// TIA Portal V17 export
// export: Created 2025-03-07T09:18:45.8638249Z, ExportSetting WithDefaults, DisplayName Totally Integrated Automation Portal, DisplayVersion V17 Update 8, DisplayName TIA Portal Openness, DisplayVersion V17 Update 8, DisplayName TIA Portal Version Control Interface, DisplayVersion V17, DisplayName SINAMICS Startdrive Advanced, DisplayVersion V17 SP2, DisplayName SINAMICS Startdrive G110M, G120, G120C, G120D, G120P, G115D, DisplayVersion V17 SP2, DisplayName SINAMICS Startdrive G130, G150, S120, S150, SINAMICS MV, S210, DisplayVersion V17 SP2, DisplayName STEP 7 Professional, DisplayVersion V17 Update 8, DisplayName SINUMERIK ONE STEP 7 Toolbox, DisplayVersion V17 Update 12, DisplayName SINUMERIK 840D sl STEP 7 Toolbox, DisplayVersion V17 Update 12, DisplayName STEP 7 Safety, DisplayVersion V17 Update 6, DisplayName WinCC Advanced, DisplayVersion V17 Update 8
FUNCTION "FC2391_SAVE_ENERGY" : Void   // FC2391, LAD
{ S7_Optimized_Access := 'FALSE' }
AUTHOR : ETXETAR
VERSION : 1.0
// stored: AutoNumber false, IsIECCheckEnabled false, SetENOAutomatically false, UDAEnableTagReadback false
   VAR_TEMP
      O_BYTE_0 : Struct   // OPTIONS BYTE 0
         AUTO_RECOVERY : Bool;   // AUTO RECOVERY OPTION
         RUNOUT : Bool;   // RUNOUT OPTION
      END_STRUCT;
   END_VAR
   VAR CONSTANT
      FC_NUMBER : DInt := 2391;
   END_VAR
   VAR_TEMP   // added for the SCL form of the ladder/FBD networks
      _w1 : Bool;
   END_VAR
BEGIN

REGION Network 1: OPTIONS OFF
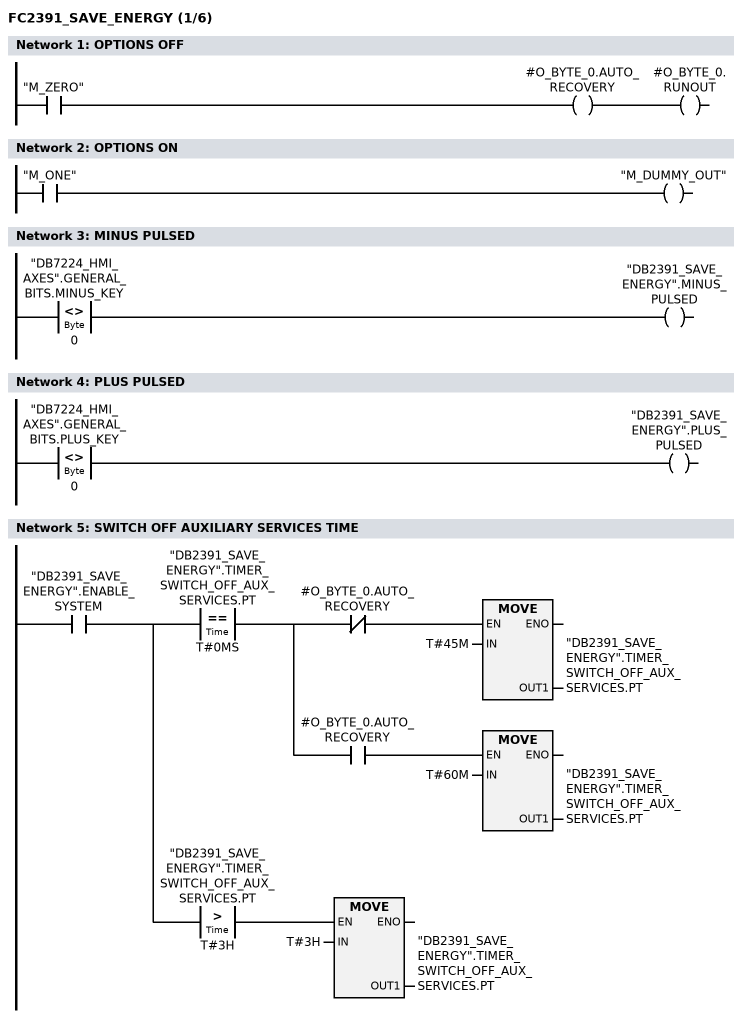
   RUNG wire#powerrail
      Contact( "M_ZERO" )
      Coil( #O_BYTE_0.AUTO_RECOVERY )
      Coil( #O_BYTE_0.RUNOUT )
   END_RUNG
   // the same network as SCL:
   #O_BYTE_0.AUTO_RECOVERY := "M_ZERO";
   #O_BYTE_0.RUNOUT := "M_ZERO";
END_REGION

REGION Network 2: OPTIONS ON
   RUNG wire#powerrail
      Contact( "M_ONE" )
      Coil( "M_DUMMY_OUT" )
   END_RUNG
   // the same network as SCL:
   "M_DUMMY_OUT" := "M_ONE";
END_REGION

REGION Network 3: MINUS PULSED
   RUNG wire#powerrail
      { S7_Templates := "SrcType := Byte" } NE_Contact(in1 := "DB7224_HMI_AXES".GENERAL_BITS.MINUS_KEY, in2 := 0)
      Coil( "DB2391_SAVE_ENERGY".MINUS_PULSED )
   END_RUNG
   // the same network as SCL:
   "DB2391_SAVE_ENERGY".MINUS_PULSED := "DB7224_HMI_AXES".GENERAL_BITS.MINUS_KEY <> 0;
END_REGION

REGION Network 4: PLUS PULSED
   RUNG wire#powerrail
      { S7_Templates := "SrcType := Byte" } NE_Contact(in1 := "DB7224_HMI_AXES".GENERAL_BITS.PLUS_KEY, in2 := 0)
      Coil( "DB2391_SAVE_ENERGY".PLUS_PULSED )
   END_RUNG
   // the same network as SCL:
   "DB2391_SAVE_ENERGY".PLUS_PULSED := "DB7224_HMI_AXES".GENERAL_BITS.PLUS_KEY <> 0;
END_REGION

REGION Network 5: SWITCH OFF AUXILIARY SERVICES TIME
   RUNG wire#powerrail
      Contact( "DB2391_SAVE_ENERGY".ENABLE_SYSTEM )
      wire#w1
      { S7_Templates := "SrcType := Time" } EQ_Contact(in1 := "DB2391_SAVE_ENERGY".TIMER_SWITCH_OFF_AUX_SERVICES.PT, in2 := T#0MS)
      wire#w2
      I_Contact( #O_BYTE_0.AUTO_RECOVERY )
      { S7_GenerateENO := "TRUE" } Move(in := T#45M, out1 => "DB2391_SAVE_ENERGY".TIMER_SWITCH_OFF_AUX_SERVICES.PT)
   END_RUNG
   RUNG wire#w2
      Contact( #O_BYTE_0.AUTO_RECOVERY )
      { S7_GenerateENO := "TRUE" } Move(in := T#60M, out1 => "DB2391_SAVE_ENERGY".TIMER_SWITCH_OFF_AUX_SERVICES.PT)
   END_RUNG
   RUNG wire#w1
      { S7_Templates := "SrcType := Time" } GT_Contact(in1 := "DB2391_SAVE_ENERGY".TIMER_SWITCH_OFF_AUX_SERVICES.PT, in2 := T#3H)
      { S7_GenerateENO := "TRUE" } Move(in := T#3H, out1 => "DB2391_SAVE_ENERGY".TIMER_SWITCH_OFF_AUX_SERVICES.PT)
   END_RUNG
   // the same network as SCL:
   #_w1 := "DB2391_SAVE_ENERGY".ENABLE_SYSTEM AND ("DB2391_SAVE_ENERGY".TIMER_SWITCH_OFF_AUX_SERVICES.PT = T#0MS);
   IF #_w1 AND NOT #O_BYTE_0.AUTO_RECOVERY THEN
       "DB2391_SAVE_ENERGY".TIMER_SWITCH_OFF_AUX_SERVICES.PT := T#45M;
   END_IF;
   IF #_w1 AND #O_BYTE_0.AUTO_RECOVERY THEN
       "DB2391_SAVE_ENERGY".TIMER_SWITCH_OFF_AUX_SERVICES.PT := T#60M;
   END_IF;
   IF "DB2391_SAVE_ENERGY".ENABLE_SYSTEM AND ("DB2391_SAVE_ENERGY".TIMER_SWITCH_OFF_AUX_SERVICES.PT > T#3H) THEN
       "DB2391_SAVE_ENERGY".TIMER_SWITCH_OFF_AUX_SERVICES.PT := T#3H;
   END_IF;
END_REGION

REGION Network 6: SWITCH OFF MAIN SERVICES TIME
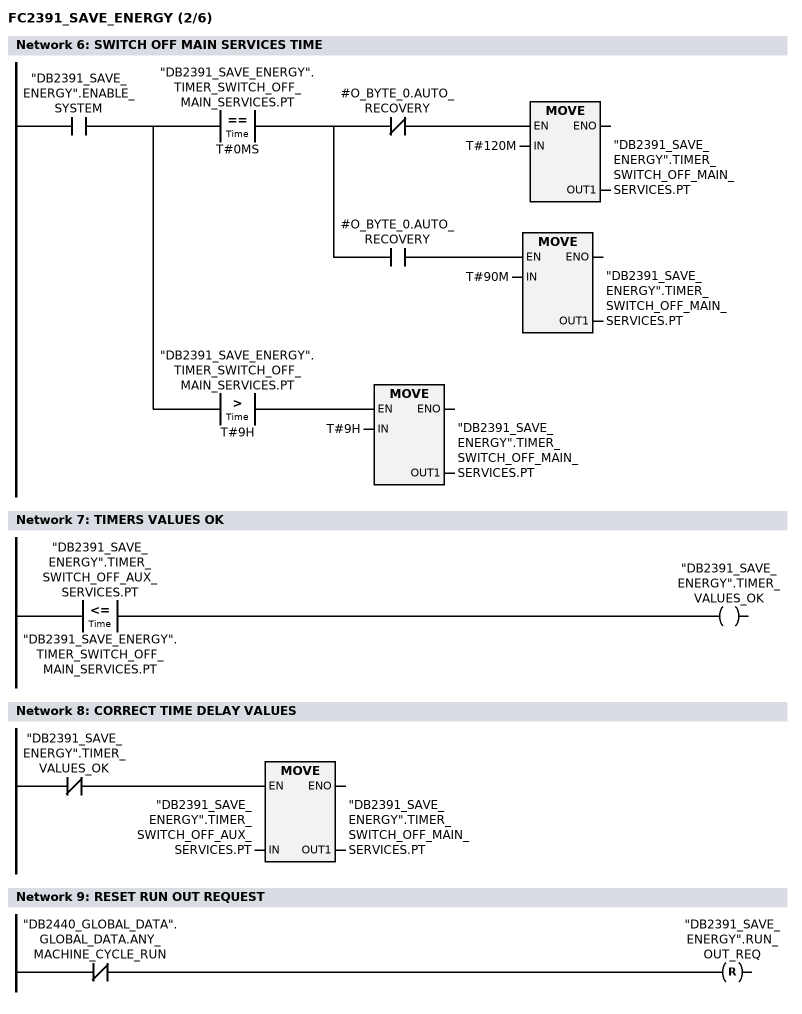
   RUNG wire#powerrail
      Contact( "DB2391_SAVE_ENERGY".ENABLE_SYSTEM )
      wire#w1
      { S7_Templates := "SrcType := Time" } EQ_Contact(in1 := "DB2391_SAVE_ENERGY".TIMER_SWITCH_OFF_MAIN_SERVICES.PT, in2 := T#0MS)
      wire#w2
      I_Contact( #O_BYTE_0.AUTO_RECOVERY )
      { S7_GenerateENO := "TRUE" } Move(in := T#120M, out1 => "DB2391_SAVE_ENERGY".TIMER_SWITCH_OFF_MAIN_SERVICES.PT)
   END_RUNG
   RUNG wire#w2
      Contact( #O_BYTE_0.AUTO_RECOVERY )
      { S7_GenerateENO := "TRUE" } Move(in := T#90M, out1 => "DB2391_SAVE_ENERGY".TIMER_SWITCH_OFF_MAIN_SERVICES.PT)
   END_RUNG
   RUNG wire#w1
      { S7_Templates := "SrcType := Time" } GT_Contact(in1 := "DB2391_SAVE_ENERGY".TIMER_SWITCH_OFF_MAIN_SERVICES.PT, in2 := T#9H)
      { S7_GenerateENO := "TRUE" } Move(in := T#9H, out1 => "DB2391_SAVE_ENERGY".TIMER_SWITCH_OFF_MAIN_SERVICES.PT)
   END_RUNG
   // the same network as SCL:
   #_w1 := "DB2391_SAVE_ENERGY".ENABLE_SYSTEM AND ("DB2391_SAVE_ENERGY".TIMER_SWITCH_OFF_MAIN_SERVICES.PT = T#0MS);
   IF #_w1 AND NOT #O_BYTE_0.AUTO_RECOVERY THEN
       "DB2391_SAVE_ENERGY".TIMER_SWITCH_OFF_MAIN_SERVICES.PT := T#120M;
   END_IF;
   IF #_w1 AND #O_BYTE_0.AUTO_RECOVERY THEN
       "DB2391_SAVE_ENERGY".TIMER_SWITCH_OFF_MAIN_SERVICES.PT := T#90M;
   END_IF;
   IF "DB2391_SAVE_ENERGY".ENABLE_SYSTEM AND ("DB2391_SAVE_ENERGY".TIMER_SWITCH_OFF_MAIN_SERVICES.PT > T#9H) THEN
       "DB2391_SAVE_ENERGY".TIMER_SWITCH_OFF_MAIN_SERVICES.PT := T#9H;
   END_IF;
END_REGION

REGION Network 7: TIMERS VALUES OK
   RUNG wire#powerrail
      { S7_Templates := "SrcType := Time" } LE_Contact(in1 := "DB2391_SAVE_ENERGY".TIMER_SWITCH_OFF_AUX_SERVICES.PT, in2 := "DB2391_SAVE_ENERGY".TIMER_SWITCH_OFF_MAIN_SERVICES.PT)
      Coil( "DB2391_SAVE_ENERGY".TIMER_VALUES_OK )
   END_RUNG
   // the same network as SCL:
   "DB2391_SAVE_ENERGY".TIMER_VALUES_OK := "DB2391_SAVE_ENERGY".TIMER_SWITCH_OFF_AUX_SERVICES.PT <= "DB2391_SAVE_ENERGY".TIMER_SWITCH_OFF_MAIN_SERVICES.PT;
END_REGION

REGION Network 8: CORRECT TIME DELAY VALUES
   RUNG wire#powerrail
      I_Contact( "DB2391_SAVE_ENERGY".TIMER_VALUES_OK )
      Move(in := "DB2391_SAVE_ENERGY".TIMER_SWITCH_OFF_AUX_SERVICES.PT, out1 => "DB2391_SAVE_ENERGY".TIMER_SWITCH_OFF_MAIN_SERVICES.PT)
   END_RUNG
   // the same network as SCL:
   IF NOT "DB2391_SAVE_ENERGY".TIMER_VALUES_OK THEN
       "DB2391_SAVE_ENERGY".TIMER_SWITCH_OFF_MAIN_SERVICES.PT := "DB2391_SAVE_ENERGY".TIMER_SWITCH_OFF_AUX_SERVICES.PT;
   END_IF;
END_REGION

REGION Network 9: RESET RUN OUT REQUEST
   RUNG wire#powerrail
      I_Contact( "DB2440_GLOBAL_DATA".GLOBAL_DATA.ANY_MACHINE_CYCLE_RUN )
      R_Coil( "DB2391_SAVE_ENERGY".RUN_OUT_REQ )
   END_RUNG
   // the same network as SCL:
   IF NOT "DB2440_GLOBAL_DATA".GLOBAL_DATA.ANY_MACHINE_CYCLE_RUN THEN
       "DB2391_SAVE_ENERGY".RUN_OUT_REQ := FALSE;
   END_IF;
END_REGION

REGION Network 10: RUN OUT REQUEST
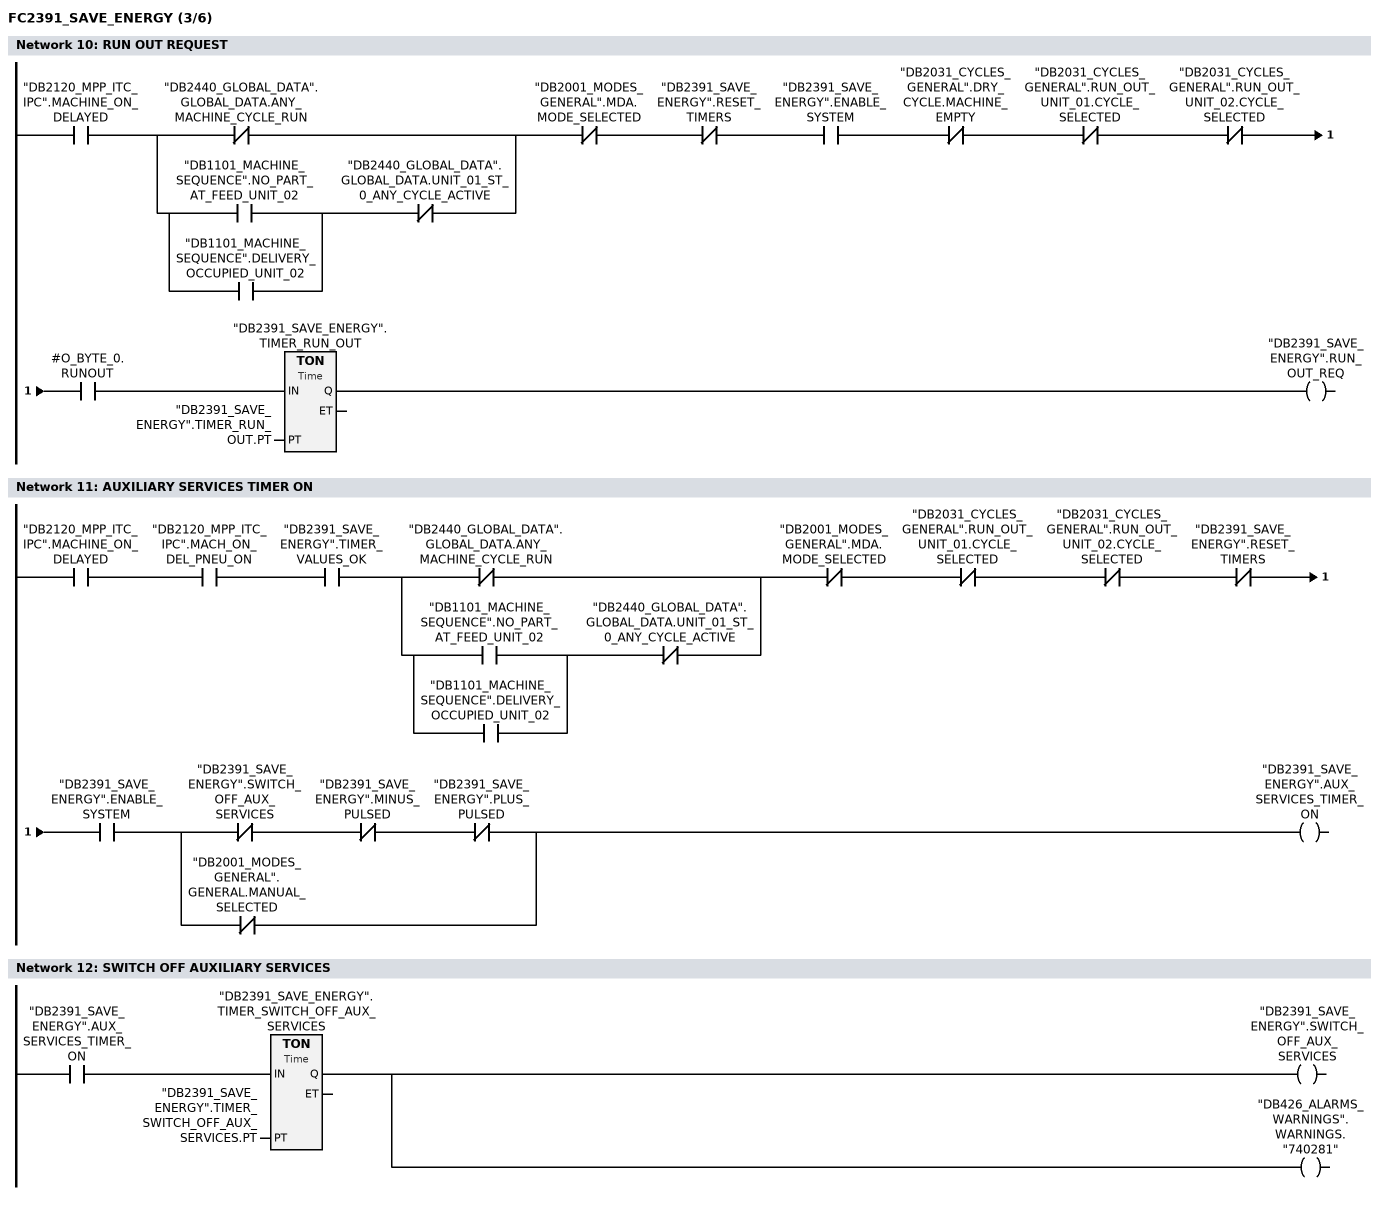
   RUNG wire#powerrail
      Contact( "DB2120_MPP_ITC_IPC".MACHINE_ON_DELAYED )
      wire#w1
      I_Contact( "DB2440_GLOBAL_DATA".GLOBAL_DATA.ANY_MACHINE_CYCLE_RUN )
      wire#w2
      I_Contact( "DB2001_MODES_GENERAL".MDA.MODE_SELECTED )
      I_Contact( "DB2391_SAVE_ENERGY".RESET_TIMERS )
      Contact( "DB2391_SAVE_ENERGY".ENABLE_SYSTEM )
      I_Contact( "DB2031_CYCLES_GENERAL".DRY_CYCLE.MACHINE_EMPTY )
      I_Contact( "DB2031_CYCLES_GENERAL".RUN_OUT_UNIT_01.CYCLE_SELECTED )
      I_Contact( "DB2031_CYCLES_GENERAL".RUN_OUT_UNIT_02.CYCLE_SELECTED )
      Contact( #O_BYTE_0.RUNOUT )
      { S7_Templates := "time_type := Time" } "DB2391_SAVE_ENERGY".TIMER_RUN_OUT.TON(pt := "DB2391_SAVE_ENERGY".TIMER_RUN_OUT.PT, et =>)
      Coil( "DB2391_SAVE_ENERGY".RUN_OUT_REQ )
   END_RUNG
   RUNG wire#w1
      Contact( "DB1101_MACHINE_SEQUENCE".NO_PART_AT_FEED_UNIT_02 )
      wire#w3
      I_Contact( "DB2440_GLOBAL_DATA".GLOBAL_DATA.UNIT_01_ST_0_ANY_CYCLE_ACTIVE )
   END_RUNG wire#w2
   RUNG wire#w1
      Contact( "DB1101_MACHINE_SEQUENCE".DELIVERY_OCCUPIED_UNIT_02 )
   END_RUNG wire#w3
   // the same network as SCL:
   "DB2391_SAVE_ENERGY".TIMER_RUN_OUT.TON(IN := "DB2120_MPP_ITC_IPC".MACHINE_ON_DELAYED AND (NOT "DB2440_GLOBAL_DATA".GLOBAL_DATA.ANY_MACHINE_CYCLE_RUN OR (("DB1101_MACHINE_SEQUENCE".NO_PART_AT_FEED_UNIT_02 OR "DB1101_MACHINE_SEQUENCE".DELIVERY_OCCUPIED_UNIT_02) AND NOT "DB2440_GLOBAL_DATA".GLOBAL_DATA.UNIT_01_ST_0_ANY_CYCLE_ACTIVE)) AND NOT "DB2001_MODES_GENERAL".MDA.MODE_SELECTED AND NOT "DB2391_SAVE_ENERGY".RESET_TIMERS AND "DB2391_SAVE_ENERGY".ENABLE_SYSTEM AND NOT "DB2031_CYCLES_GENERAL".DRY_CYCLE.MACHINE_EMPTY AND NOT "DB2031_CYCLES_GENERAL".RUN_OUT_UNIT_01.CYCLE_SELECTED AND NOT "DB2031_CYCLES_GENERAL".RUN_OUT_UNIT_02.CYCLE_SELECTED AND #O_BYTE_0.RUNOUT,
                           PT := "DB2391_SAVE_ENERGY".TIMER_RUN_OUT.PT);
   "DB2391_SAVE_ENERGY".RUN_OUT_REQ := "DB2391_SAVE_ENERGY".TIMER_RUN_OUT.Q;
END_REGION

REGION Network 11: AUXILIARY SERVICES TIMER ON
   RUNG wire#powerrail
      Contact( "DB2120_MPP_ITC_IPC".MACHINE_ON_DELAYED )
      Contact( "DB2120_MPP_ITC_IPC".MACH_ON_DEL_PNEU_ON )
      Contact( "DB2391_SAVE_ENERGY".TIMER_VALUES_OK )
      wire#w1
      I_Contact( "DB2440_GLOBAL_DATA".GLOBAL_DATA.ANY_MACHINE_CYCLE_RUN )
      wire#w2
      I_Contact( "DB2001_MODES_GENERAL".MDA.MODE_SELECTED )
      I_Contact( "DB2031_CYCLES_GENERAL".RUN_OUT_UNIT_01.CYCLE_SELECTED )
      I_Contact( "DB2031_CYCLES_GENERAL".RUN_OUT_UNIT_02.CYCLE_SELECTED )
      I_Contact( "DB2391_SAVE_ENERGY".RESET_TIMERS )
      Contact( "DB2391_SAVE_ENERGY".ENABLE_SYSTEM )
      wire#w4
      I_Contact( "DB2391_SAVE_ENERGY".SWITCH_OFF_AUX_SERVICES )
      I_Contact( "DB2391_SAVE_ENERGY".MINUS_PULSED )
      I_Contact( "DB2391_SAVE_ENERGY".PLUS_PULSED )
      wire#w5
      Coil( "DB2391_SAVE_ENERGY".AUX_SERVICES_TIMER_ON )
   END_RUNG
   RUNG wire#w1
      Contact( "DB1101_MACHINE_SEQUENCE".NO_PART_AT_FEED_UNIT_02 )
      wire#w3
      I_Contact( "DB2440_GLOBAL_DATA".GLOBAL_DATA.UNIT_01_ST_0_ANY_CYCLE_ACTIVE )
   END_RUNG wire#w2
   RUNG wire#w1
      Contact( "DB1101_MACHINE_SEQUENCE".DELIVERY_OCCUPIED_UNIT_02 )
   END_RUNG wire#w3
   RUNG wire#w4
      I_Contact( "DB2001_MODES_GENERAL".GENERAL.MANUAL_SELECTED )
   END_RUNG wire#w5
   // the same network as SCL:
   "DB2391_SAVE_ENERGY".AUX_SERVICES_TIMER_ON := "DB2120_MPP_ITC_IPC".MACHINE_ON_DELAYED AND "DB2120_MPP_ITC_IPC".MACH_ON_DEL_PNEU_ON AND "DB2391_SAVE_ENERGY".TIMER_VALUES_OK AND (NOT "DB2440_GLOBAL_DATA".GLOBAL_DATA.ANY_MACHINE_CYCLE_RUN OR (("DB1101_MACHINE_SEQUENCE".NO_PART_AT_FEED_UNIT_02 OR "DB1101_MACHINE_SEQUENCE".DELIVERY_OCCUPIED_UNIT_02) AND NOT "DB2440_GLOBAL_DATA".GLOBAL_DATA.UNIT_01_ST_0_ANY_CYCLE_ACTIVE)) AND NOT "DB2001_MODES_GENERAL".MDA.MODE_SELECTED AND NOT "DB2031_CYCLES_GENERAL".RUN_OUT_UNIT_01.CYCLE_SELECTED AND NOT "DB2031_CYCLES_GENERAL".RUN_OUT_UNIT_02.CYCLE_SELECTED AND NOT "DB2391_SAVE_ENERGY".RESET_TIMERS AND "DB2391_SAVE_ENERGY".ENABLE_SYSTEM AND ((NOT "DB2391_SAVE_ENERGY".SWITCH_OFF_AUX_SERVICES AND NOT "DB2391_SAVE_ENERGY".MINUS_PULSED AND NOT "DB2391_SAVE_ENERGY".PLUS_PULSED) OR NOT "DB2001_MODES_GENERAL".GENERAL.MANUAL_SELECTED);
END_REGION

REGION Network 12: SWITCH OFF AUXILIARY SERVICES
   RUNG wire#powerrail
      Contact( "DB2391_SAVE_ENERGY".AUX_SERVICES_TIMER_ON )
      { S7_Templates := "time_type := Time" } "DB2391_SAVE_ENERGY".TIMER_SWITCH_OFF_AUX_SERVICES.TON(pt := "DB2391_SAVE_ENERGY".TIMER_SWITCH_OFF_AUX_SERVICES.PT, et =>)
      wire#w1
      Coil( "DB2391_SAVE_ENERGY".SWITCH_OFF_AUX_SERVICES )
   END_RUNG
   RUNG wire#w1
      Coil( "DB426_ALARMS_WARNINGS".WARNINGS."740281" )
   END_RUNG
   // the same network as SCL:
   "DB2391_SAVE_ENERGY".TIMER_SWITCH_OFF_AUX_SERVICES.TON(IN := "DB2391_SAVE_ENERGY".AUX_SERVICES_TIMER_ON,
                           PT := "DB2391_SAVE_ENERGY".TIMER_SWITCH_OFF_AUX_SERVICES.PT);
   "DB2391_SAVE_ENERGY".SWITCH_OFF_AUX_SERVICES := "DB2391_SAVE_ENERGY".TIMER_SWITCH_OFF_AUX_SERVICES.Q;
   "DB426_ALARMS_WARNINGS".WARNINGS."740281" := "DB2391_SAVE_ENERGY".TIMER_SWITCH_OFF_AUX_SERVICES.Q;
END_REGION

REGION Network 13: SWTICH OFF AUXILIARY SERVICES TIME LEFT
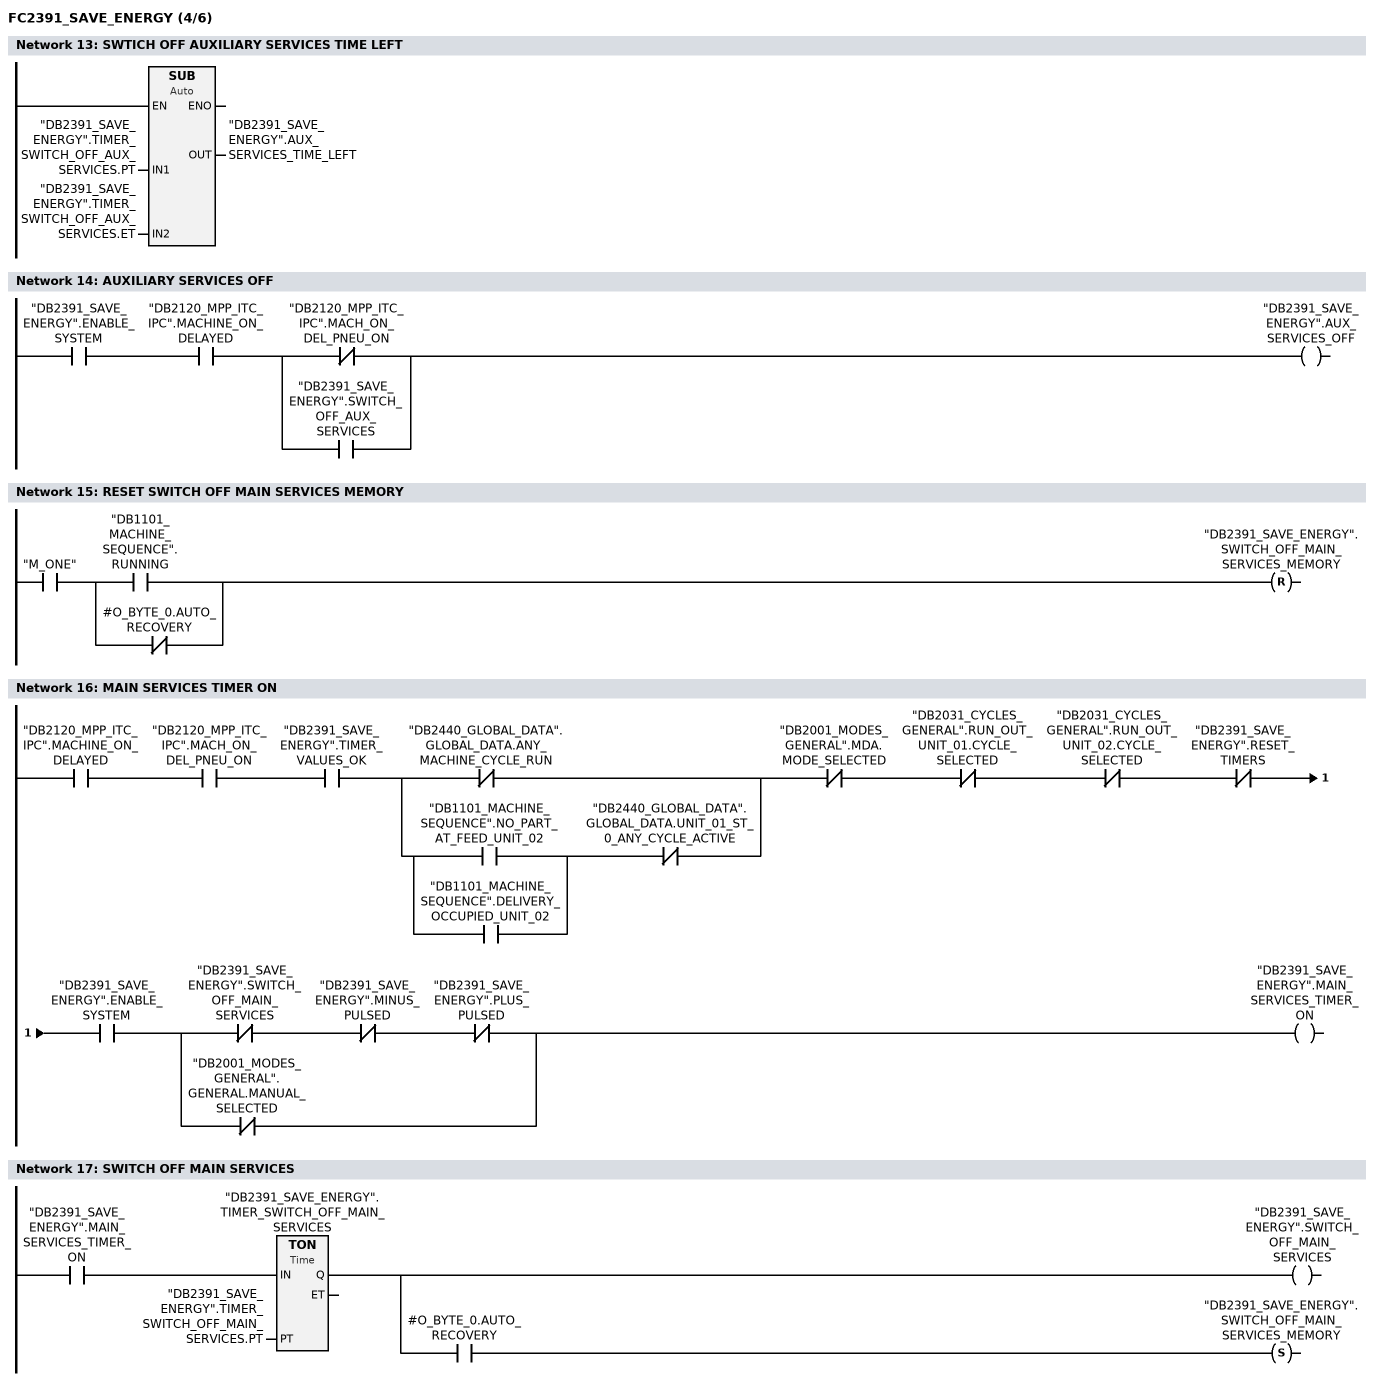
   RUNG wire#powerrail
      Sub(in1 := "DB2391_SAVE_ENERGY".TIMER_SWITCH_OFF_AUX_SERVICES.PT, in2 := "DB2391_SAVE_ENERGY".TIMER_SWITCH_OFF_AUX_SERVICES.ET, out => "DB2391_SAVE_ENERGY".AUX_SERVICES_TIME_LEFT)
   END_RUNG
   // the same network as SCL:
   "DB2391_SAVE_ENERGY".AUX_SERVICES_TIME_LEFT := "DB2391_SAVE_ENERGY".TIMER_SWITCH_OFF_AUX_SERVICES.PT - "DB2391_SAVE_ENERGY".TIMER_SWITCH_OFF_AUX_SERVICES.ET;
END_REGION

REGION Network 14: AUXILIARY SERVICES OFF
   RUNG wire#powerrail
      Contact( "DB2391_SAVE_ENERGY".ENABLE_SYSTEM )
      Contact( "DB2120_MPP_ITC_IPC".MACHINE_ON_DELAYED )
      wire#w1
      I_Contact( "DB2120_MPP_ITC_IPC".MACH_ON_DEL_PNEU_ON )
      wire#w2
      Coil( "DB2391_SAVE_ENERGY".AUX_SERVICES_OFF )
   END_RUNG
   RUNG wire#w1
      Contact( "DB2391_SAVE_ENERGY".SWITCH_OFF_AUX_SERVICES )
   END_RUNG wire#w2
   // the same network as SCL:
   "DB2391_SAVE_ENERGY".AUX_SERVICES_OFF := "DB2391_SAVE_ENERGY".ENABLE_SYSTEM AND "DB2120_MPP_ITC_IPC".MACHINE_ON_DELAYED AND (NOT "DB2120_MPP_ITC_IPC".MACH_ON_DEL_PNEU_ON OR "DB2391_SAVE_ENERGY".SWITCH_OFF_AUX_SERVICES);
END_REGION

REGION Network 15: RESET SWITCH OFF MAIN SERVICES MEMORY
   RUNG wire#powerrail
      Contact( "M_ONE" )
      wire#w1
      Contact( "DB1101_MACHINE_SEQUENCE".RUNNING )
      wire#w2
      R_Coil( "DB2391_SAVE_ENERGY".SWITCH_OFF_MAIN_SERVICES_MEMORY )
   END_RUNG
   RUNG wire#w1
      I_Contact( #O_BYTE_0.AUTO_RECOVERY )
   END_RUNG wire#w2
   // the same network as SCL:
   IF "M_ONE" AND ("DB1101_MACHINE_SEQUENCE".RUNNING OR NOT #O_BYTE_0.AUTO_RECOVERY) THEN
       "DB2391_SAVE_ENERGY".SWITCH_OFF_MAIN_SERVICES_MEMORY := FALSE;
   END_IF;
END_REGION

REGION Network 16: MAIN SERVICES TIMER ON
   RUNG wire#powerrail
      Contact( "DB2120_MPP_ITC_IPC".MACHINE_ON_DELAYED )
      Contact( "DB2120_MPP_ITC_IPC".MACH_ON_DEL_PNEU_ON )
      Contact( "DB2391_SAVE_ENERGY".TIMER_VALUES_OK )
      wire#w1
      I_Contact( "DB2440_GLOBAL_DATA".GLOBAL_DATA.ANY_MACHINE_CYCLE_RUN )
      wire#w2
      I_Contact( "DB2001_MODES_GENERAL".MDA.MODE_SELECTED )
      I_Contact( "DB2031_CYCLES_GENERAL".RUN_OUT_UNIT_01.CYCLE_SELECTED )
      I_Contact( "DB2031_CYCLES_GENERAL".RUN_OUT_UNIT_02.CYCLE_SELECTED )
      I_Contact( "DB2391_SAVE_ENERGY".RESET_TIMERS )
      Contact( "DB2391_SAVE_ENERGY".ENABLE_SYSTEM )
      wire#w4
      I_Contact( "DB2391_SAVE_ENERGY".SWITCH_OFF_MAIN_SERVICES )
      I_Contact( "DB2391_SAVE_ENERGY".MINUS_PULSED )
      I_Contact( "DB2391_SAVE_ENERGY".PLUS_PULSED )
      wire#w5
      Coil( "DB2391_SAVE_ENERGY".MAIN_SERVICES_TIMER_ON )
   END_RUNG
   RUNG wire#w1
      Contact( "DB1101_MACHINE_SEQUENCE".NO_PART_AT_FEED_UNIT_02 )
      wire#w3
      I_Contact( "DB2440_GLOBAL_DATA".GLOBAL_DATA.UNIT_01_ST_0_ANY_CYCLE_ACTIVE )
   END_RUNG wire#w2
   RUNG wire#w1
      Contact( "DB1101_MACHINE_SEQUENCE".DELIVERY_OCCUPIED_UNIT_02 )
   END_RUNG wire#w3
   RUNG wire#w4
      I_Contact( "DB2001_MODES_GENERAL".GENERAL.MANUAL_SELECTED )
   END_RUNG wire#w5
   // the same network as SCL:
   "DB2391_SAVE_ENERGY".MAIN_SERVICES_TIMER_ON := "DB2120_MPP_ITC_IPC".MACHINE_ON_DELAYED AND "DB2120_MPP_ITC_IPC".MACH_ON_DEL_PNEU_ON AND "DB2391_SAVE_ENERGY".TIMER_VALUES_OK AND (NOT "DB2440_GLOBAL_DATA".GLOBAL_DATA.ANY_MACHINE_CYCLE_RUN OR (("DB1101_MACHINE_SEQUENCE".NO_PART_AT_FEED_UNIT_02 OR "DB1101_MACHINE_SEQUENCE".DELIVERY_OCCUPIED_UNIT_02) AND NOT "DB2440_GLOBAL_DATA".GLOBAL_DATA.UNIT_01_ST_0_ANY_CYCLE_ACTIVE)) AND NOT "DB2001_MODES_GENERAL".MDA.MODE_SELECTED AND NOT "DB2031_CYCLES_GENERAL".RUN_OUT_UNIT_01.CYCLE_SELECTED AND NOT "DB2031_CYCLES_GENERAL".RUN_OUT_UNIT_02.CYCLE_SELECTED AND NOT "DB2391_SAVE_ENERGY".RESET_TIMERS AND "DB2391_SAVE_ENERGY".ENABLE_SYSTEM AND ((NOT "DB2391_SAVE_ENERGY".SWITCH_OFF_MAIN_SERVICES AND NOT "DB2391_SAVE_ENERGY".MINUS_PULSED AND NOT "DB2391_SAVE_ENERGY".PLUS_PULSED) OR NOT "DB2001_MODES_GENERAL".GENERAL.MANUAL_SELECTED);
END_REGION

REGION Network 17: SWITCH OFF MAIN SERVICES
   RUNG wire#powerrail
      Contact( "DB2391_SAVE_ENERGY".MAIN_SERVICES_TIMER_ON )
      { S7_Templates := "time_type := Time" } "DB2391_SAVE_ENERGY".TIMER_SWITCH_OFF_MAIN_SERVICES.TON(pt := "DB2391_SAVE_ENERGY".TIMER_SWITCH_OFF_MAIN_SERVICES.PT, et =>)
      wire#w1
      Coil( "DB2391_SAVE_ENERGY".SWITCH_OFF_MAIN_SERVICES )
   END_RUNG
   RUNG wire#w1
      Contact( #O_BYTE_0.AUTO_RECOVERY )
      S_Coil( "DB2391_SAVE_ENERGY".SWITCH_OFF_MAIN_SERVICES_MEMORY )
   END_RUNG
   // the same network as SCL:
   "DB2391_SAVE_ENERGY".TIMER_SWITCH_OFF_MAIN_SERVICES.TON(IN := "DB2391_SAVE_ENERGY".MAIN_SERVICES_TIMER_ON,
                           PT := "DB2391_SAVE_ENERGY".TIMER_SWITCH_OFF_MAIN_SERVICES.PT);
   "DB2391_SAVE_ENERGY".SWITCH_OFF_MAIN_SERVICES := "DB2391_SAVE_ENERGY".TIMER_SWITCH_OFF_MAIN_SERVICES.Q;
   IF "DB2391_SAVE_ENERGY".TIMER_SWITCH_OFF_MAIN_SERVICES.Q AND #O_BYTE_0.AUTO_RECOVERY THEN
       "DB2391_SAVE_ENERGY".SWITCH_OFF_MAIN_SERVICES_MEMORY := TRUE;
   END_IF;
END_REGION

REGION Network 18: (WRN) SAVE ENERGY MAIN SERVICES OFF
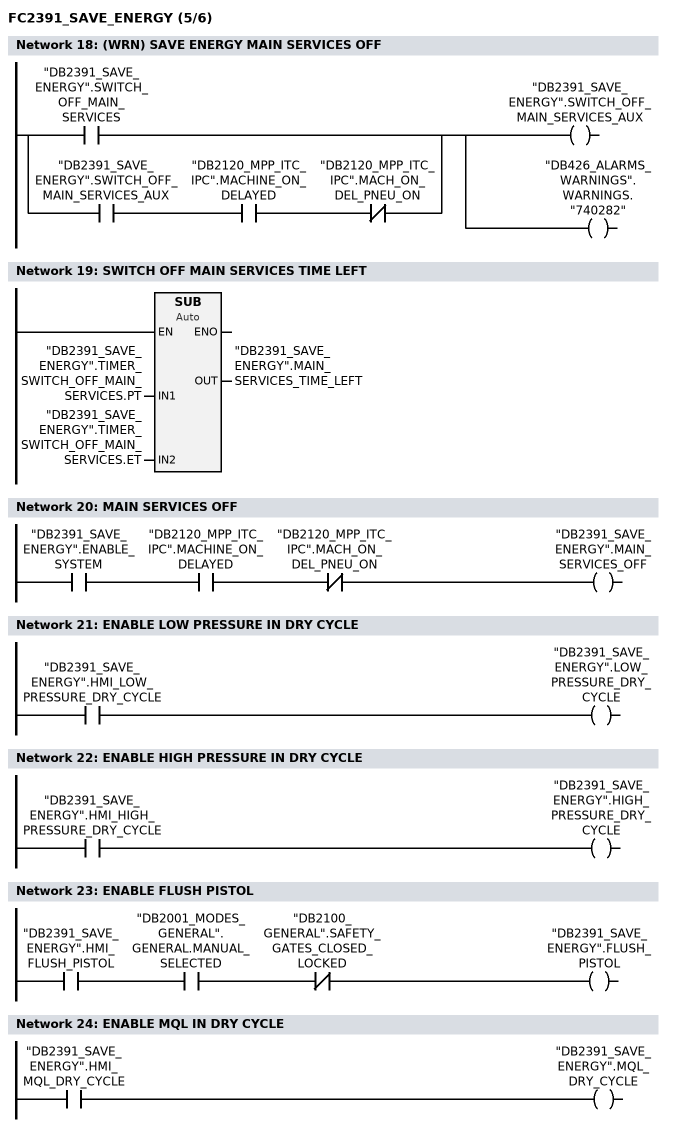
   RUNG wire#powerrail
      Contact( "DB2391_SAVE_ENERGY".SWITCH_OFF_MAIN_SERVICES )
      wire#w1
      Coil( "DB2391_SAVE_ENERGY".SWITCH_OFF_MAIN_SERVICES_AUX )
   END_RUNG
   RUNG wire#powerrail
      Contact( "DB2391_SAVE_ENERGY".SWITCH_OFF_MAIN_SERVICES_AUX )
      Contact( "DB2120_MPP_ITC_IPC".MACHINE_ON_DELAYED )
      I_Contact( "DB2120_MPP_ITC_IPC".MACH_ON_DEL_PNEU_ON )
   END_RUNG wire#w1
   RUNG wire#w1
      Coil( "DB426_ALARMS_WARNINGS".WARNINGS."740282" )
   END_RUNG
   // the same network as SCL:
   "DB2391_SAVE_ENERGY".SWITCH_OFF_MAIN_SERVICES_AUX := "DB2391_SAVE_ENERGY".SWITCH_OFF_MAIN_SERVICES OR ("DB2391_SAVE_ENERGY".SWITCH_OFF_MAIN_SERVICES_AUX AND "DB2120_MPP_ITC_IPC".MACHINE_ON_DELAYED AND NOT "DB2120_MPP_ITC_IPC".MACH_ON_DEL_PNEU_ON);
   "DB426_ALARMS_WARNINGS".WARNINGS."740282" := "DB2391_SAVE_ENERGY".SWITCH_OFF_MAIN_SERVICES_AUX;
END_REGION

REGION Network 19: SWITCH OFF MAIN SERVICES TIME LEFT
   RUNG wire#powerrail
      Sub(in1 := "DB2391_SAVE_ENERGY".TIMER_SWITCH_OFF_MAIN_SERVICES.PT, in2 := "DB2391_SAVE_ENERGY".TIMER_SWITCH_OFF_MAIN_SERVICES.ET, out => "DB2391_SAVE_ENERGY".MAIN_SERVICES_TIME_LEFT)
   END_RUNG
   // the same network as SCL:
   "DB2391_SAVE_ENERGY".MAIN_SERVICES_TIME_LEFT := "DB2391_SAVE_ENERGY".TIMER_SWITCH_OFF_MAIN_SERVICES.PT - "DB2391_SAVE_ENERGY".TIMER_SWITCH_OFF_MAIN_SERVICES.ET;
END_REGION

REGION Network 20: MAIN SERVICES OFF
   RUNG wire#powerrail
      Contact( "DB2391_SAVE_ENERGY".ENABLE_SYSTEM )
      Contact( "DB2120_MPP_ITC_IPC".MACHINE_ON_DELAYED )
      I_Contact( "DB2120_MPP_ITC_IPC".MACH_ON_DEL_PNEU_ON )
      Coil( "DB2391_SAVE_ENERGY".MAIN_SERVICES_OFF )
   END_RUNG
   // the same network as SCL:
   "DB2391_SAVE_ENERGY".MAIN_SERVICES_OFF := "DB2391_SAVE_ENERGY".ENABLE_SYSTEM AND "DB2120_MPP_ITC_IPC".MACHINE_ON_DELAYED AND NOT "DB2120_MPP_ITC_IPC".MACH_ON_DEL_PNEU_ON;
END_REGION

REGION Network 21: ENABLE LOW PRESSURE IN DRY CYCLE
   RUNG wire#powerrail
      Contact( "DB2391_SAVE_ENERGY".HMI_LOW_PRESSURE_DRY_CYCLE )
      Coil( "DB2391_SAVE_ENERGY".LOW_PRESSURE_DRY_CYCLE )
   END_RUNG
   // the same network as SCL:
   "DB2391_SAVE_ENERGY".LOW_PRESSURE_DRY_CYCLE := "DB2391_SAVE_ENERGY".HMI_LOW_PRESSURE_DRY_CYCLE;
END_REGION

REGION Network 22: ENABLE HIGH PRESSURE IN DRY CYCLE
   RUNG wire#powerrail
      Contact( "DB2391_SAVE_ENERGY".HMI_HIGH_PRESSURE_DRY_CYCLE )
      Coil( "DB2391_SAVE_ENERGY".HIGH_PRESSURE_DRY_CYCLE )
   END_RUNG
   // the same network as SCL:
   "DB2391_SAVE_ENERGY".HIGH_PRESSURE_DRY_CYCLE := "DB2391_SAVE_ENERGY".HMI_HIGH_PRESSURE_DRY_CYCLE;
END_REGION

REGION Network 23: ENABLE FLUSH PISTOL
   RUNG wire#powerrail
      Contact( "DB2391_SAVE_ENERGY".HMI_FLUSH_PISTOL )
      Contact( "DB2001_MODES_GENERAL".GENERAL.MANUAL_SELECTED )
      I_Contact( "DB2100_GENERAL".SAFETY_GATES_CLOSED_LOCKED )
      Coil( "DB2391_SAVE_ENERGY".FLUSH_PISTOL )
   END_RUNG
   // the same network as SCL:
   "DB2391_SAVE_ENERGY".FLUSH_PISTOL := "DB2391_SAVE_ENERGY".HMI_FLUSH_PISTOL AND "DB2001_MODES_GENERAL".GENERAL.MANUAL_SELECTED AND NOT "DB2100_GENERAL".SAFETY_GATES_CLOSED_LOCKED;
END_REGION

REGION Network 24: ENABLE MQL IN DRY CYCLE
   RUNG wire#powerrail
      Contact( "DB2391_SAVE_ENERGY".HMI_MQL_DRY_CYCLE )
      Coil( "DB2391_SAVE_ENERGY".MQL_DRY_CYCLE )
   END_RUNG
   // the same network as SCL:
   "DB2391_SAVE_ENERGY".MQL_DRY_CYCLE := "DB2391_SAVE_ENERGY".HMI_MQL_DRY_CYCLE;
END_REGION

REGION Network 25: RESET HMI SETTINGS
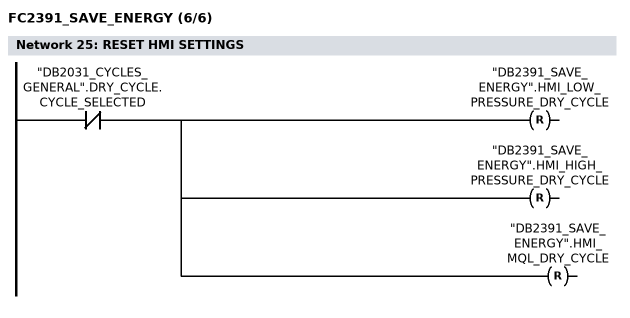
   RUNG wire#powerrail
      I_Contact( "DB2031_CYCLES_GENERAL".DRY_CYCLE.CYCLE_SELECTED )
      wire#w1
      R_Coil( "DB2391_SAVE_ENERGY".HMI_LOW_PRESSURE_DRY_CYCLE )
   END_RUNG
   RUNG wire#w1
      R_Coil( "DB2391_SAVE_ENERGY".HMI_HIGH_PRESSURE_DRY_CYCLE )
   END_RUNG
   RUNG wire#w1
      R_Coil( "DB2391_SAVE_ENERGY".HMI_MQL_DRY_CYCLE )
   END_RUNG
   // the same network as SCL:
   IF NOT "DB2031_CYCLES_GENERAL".DRY_CYCLE.CYCLE_SELECTED THEN
       "DB2391_SAVE_ENERGY".HMI_LOW_PRESSURE_DRY_CYCLE := FALSE;
       "DB2391_SAVE_ENERGY".HMI_HIGH_PRESSURE_DRY_CYCLE := FALSE;
       "DB2391_SAVE_ENERGY".HMI_MQL_DRY_CYCLE := FALSE;
   END_IF;
END_REGION
END_FUNCTION
